FUNCTION_BLOCK CoolingUnit_eChiller EXTENDS FB_ActorContinous
VAR_INPUT
	fExternalTemperature : REAL; //External temperature in °C
END_VAR
VAR_OUTPUT
	bError : BOOL; // Returns eChiller error
END_VAR
VAR
	//default parameters
	localDefaultParameters : ST_eChillerDefaultParameters;

	{attribute 'OPC.UA.DA' := '1'}
	localState : ST_PumpGrundfosMagna3State;
	
	//analog converters
	OutputConverter_SetpointValue : FB_AnalogOutput := (fUpperLimit := 28, fLowerLimit := 10);
	OutputConverter_ActualTemperature : FB_AnalogOutput := (fUpperLimit := 28, fLowerLimit := 10);
	
	//I/O Links
	nSetPoint_OUT			AT %Q* : INT; //Set position linked to terminal
	nActualTemperature_OUT 	AT %Q* : INT; //Actual temperature in buffer storage linked to terminal
	bSetStatusOn_OUT 		AT %Q* : BOOL; //SetStatus linked to terminal
	//bEmergencyStop_OUT 		AT %Q* : BOOL; //External triggered emergency stop linked to terminal - Needed?
	bError_IN 				AT %I* : BOOL; //Error state linked to terminal
	bWarning_IN 			AT %I* : BOOL; //Warning state linked to terminal
	bStatusOn_IN 			AT %I* : BOOL; //Working state linked to terminal
END_VAR

MAIN();

METHOD SetState : BOOL
VAR_INPUT
END_VAR
//control state
controlState.bStatusOn := bStatusOn_IN;

//setpoint state
setPointState.fSetPoint := fSetPoint;
setPointState.sSetPointUnit := 'degreeC';
setPointState.fOperatingPoint := fExternalTemperature;
setPointState.sOperatingPointUnit := 'degreeC';
setPointState.aSetPointLimits := aSetPointLimits;

//local state
bError := bError_IN;
localState.bError := bError_IN;
localState.bWarning := bWarning_IN;
//local state is read via opc ua

//outputs
nSetPoint_OUT := OutputConverter_SetpointValue(fValue := fSetPoint);
nActualTemperature_OUT := OutputConverter_ActualTemperature(fValue := fExternalTemperature);
bSetStatusOn_OUT := bSetStatusOn;
END_METHOD

PROPERTY ST_DefaultParameters : REFERENCE TO ST_eChillerDefaultParameters
SET
localDefaultParameters := ST_DefaultParameters;
END_SET
END_PROPERTY

END_FUNCTION_BLOCK

(* stored: Version 1.1.0.1, ProductVersion 3.1.4024.9
   POU CoolingUnit_eChiller: Id {2fd4228b-5aa5-47c8-816c-daa5107a89d5}, SpecialFunc None
   Method SetState: Id {9359ead8-ac36-4230-8c6e-96a2110ee420}
   Property ST_DefaultParameters: Id {96545930-9036-4902-a3c8-00c527dc6dce}
   Set Set: Id {45f955fa-610f-44eb-8e32-a0a25e0099c9} *)
